(* IEC 61131-3 sources: mp-conveyorbelt/src, 4 files *)

(* ---- Belt.st ---- *)
NAMESPACE Simatic.Ax.Mp
    CLASS Belt
        VAR PUBLIC
            isRunning : INT;    // 0: stopped, 1: forward, -1: backwards
            isStopped : BOOL;   // True if belt is stopped
        END_VAR
        VAR PRIVATE
            _beltData : types.beltData;     // Store belt data internally
        END_VAR

        METHOD PUBLIC RunForward
            isRunning := THIS.getSpeedSP();
            isStopped := FALSE;
        END_METHOD
        METHOD PUBLIC RunBackward
            isRunning := -1 * THIS.getSpeedSP();
            isStopped := FALSE;
        END_METHOD
        METHOD PUBLIC Stop
            isRunning := 0;
            isStopped := TRUE;
        END_METHOD

        /// GET / SET Belt-Data
        METHOD PUBLIC setBeltData
            VAR_INPUT
                beltData : types.beltData;
            END_VAR
            _beltData := beltData;
        END_METHOD

        METHOD PUBLIC getBeltData : types.beltData
            getBeltData := _beltData;
        END_METHOD

        /// GET / SET Speed
        METHOD PRIVATE getSpeedSP : INT
            getSpeedSP := _beltData.speedSP;
        END_METHOD
        METHOD PUBLIC setSpeedSP
            VAR_INPUT
                speedSP : INT;
            END_VAR

            IF speedSP >= _beltData.minSpeed AND speedSP <= _beltData.maxSpeed THEN
                _beltData.speedSP := speedSP;
            END_IF;
        END_METHOD
    END_CLASS
END_NAMESPACE

(* ---- conveyorbelt.st ---- *)
NAMESPACE Simatic.Ax.Mp

    {axcode:docs-v0:@simatic-ax/mp-conveyorbelt:conveyorbelt-class.md}
    /// This class is for demonstration purpose only
    CLASS ConveyorBelt

        VAR PUBLIC
        END_VAR

        VAR
        END_VAR

        /// Call this in order to :
        /// initialize the beltconveyor
        METHOD PUBLIC Init
            ;
        END_METHOD

        /// Call this in order to :
        /// move the conveyorbelt forward (1) with a static velocity
        METHOD PUBLIC MoveForward
            ;
        END_METHOD

        /// Call this in order to :
        /// move the conveyorbelt backward (0) with a static velocity
        METHOD PUBLIC MoveBackward
            ;
        END_METHOD

        // Call this in order to :
        /// move the conveyorbelt backward (0) with a static velocity
        METHOD PUBLIC MoveToSensor
            ;
        END_METHOD

    END_CLASS

END_NAMESPACE

(* ---- Conveyors.st ---- *)
NAMESPACE Simatic.Ax.Mp
   // Conveyors with only one belt
   CLASS OneBeltConveyor IMPLEMENTS IConveyor
      VAR PUBLIC
         belt : REF_TO Belt;
         isOn : BOOL;
      END_VAR

      METHOD PUBLIC Run
         belt^.RunForward();
         isOn := TRUE;
      END_METHOD

      METHOD PUBLIC Stop
         belt^.Stop();
         isOn := FALSE;
      END_METHOD
   END_CLASS

   // Two conveyors - one running forwards, the other one backwards
   CLASS TwoBeltConveyor IMPLEMENTS IConveyor
      VAR PUBLIC
         belt1 : REF_TO Belt;
         belt2 : REF_TO Belt;
         isOn : BOOL;
      END_VAR

      METHOD PUBLIC Run
         belt1^.RunForward();
         belt2^.RunBackward();
         isOn := TRUE;
      END_METHOD

      METHOD PUBLIC Stop
         belt1^.Stop();
         belt2^.Stop();
         isOn := FALSE;
      END_METHOD
   END_CLASS
END_NAMESPACE

(* ---- myClass.st ---- *)
NAMESPACE Simatic.Ax.Library

    {axcode:docs-v0:@simatic-ax/mp-conveyorbelt:MyClass.md}
    CLASS MyClass

        VAR PUBLIC
        END_VAR

        VAR
        END_VAR

        /// Inline Comment for MyMethod. It will be shown, when you hover over the method
        /// This method has no parameters and no return value
        METHOD PUBLIC MyMethod
            ;
        END_METHOD

    END_CLASS

END_NAMESPACE
